FUNCTION_BLOCK HMI
VAR_INPUT
END_VAR
VAR_OUTPUT
END_VAR
VAR
	wDeviceAddress : WORD;
	wMotorAddress : WORD;
	bMotorPower : BOOL;
	bMotorOvercurrent : BOOL;
	rMotorTemperature : REAL;
	rMotorSpeed : REAL;
	rMotorPosition : REAL;
END_VAR

METHOD displayValues
VAR_INPUT
END_VAR
END_METHOD

METHOD FB_init : BOOL
VAR_INPUT
	bInitRetains : BOOL; // if TRUE, the retain variables are initialized (warm start / cold start)
	bInCopyCode : BOOL;  // if TRUE, the instance afterwards gets moved into the copy code (online change)
END_VAR
END_METHOD

METHOD writeValuesToDevice : BOOL
VAR_INPUT
END_VAR
END_METHOD

END_FUNCTION_BLOCK

(* stored: Version 1.1.0.1, ProductVersion 3.1.4024.12
   POU HMI: Id {f38ad59a-78b0-4789-8887-833d8ba3ce26}, SpecialFunc None
   Method displayValues: Id {84f98107-3448-48e8-a3ae-474257ac1426}
   Method FB_init: Id {000d9a1f-0032-4f6d-a4be-ae7b9bc444e5}
   Method writeValuesToDevice: Id {803aefaf-436f-4700-a6da-a452b20c6909} *)
